FUNCTION_BLOCK FbGSS (* Генератор сигналов и псевдослучайных чисел. *)
  (* Standard: 61499-1; Description: Генератор сигналов и псевдослучайных чисел. Simple FB with one algorithm *)
  (* Version 2.1, 2026-03-20, VA, LIB_PLC *)
  (* Documentation:
  // Генератор сигналов и псевдослучайных чисел. //             DbGSS //     +--------------------+ //     |       FbGSS        | //    -|Amplitude       Sine|->- //    -|Period        Cosine|->- //    -|Phase     RectangleR|->- //    -|Offset    RectangleB|->- //    -|PulseTime   Triangle|->- //    -|Ts              Prnd|->- //     +--------------------+
  *)
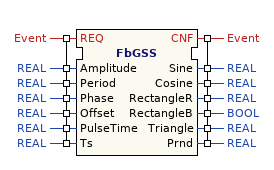
  EVENT_INPUT
    REQ WITH Amplitude, Period, Phase, Offset, PulseTime, Ts; (* Normal Execution Request *)
  END_EVENT
  EVENT_OUTPUT
    CNF WITH Sine, Cosine, RectangleR, RectangleB, Triangle, Prnd; (* Execution Confirmation *)
  END_EVENT
  VAR_INPUT
    Amplitude : REAL := 1.0; (* Амплитуда выходного сигнала. *)
    Period : REAL := 10.0; (* Период выходного сигнала [с]. *)
    Phase : REAL := 0.0; (* Фаза выходного сигнала [рад]. *)
    Offset : REAL := 0.0; (* Постоянная составляющая выходного сигнала. *)
    PulseTime : REAL := 5.0; (* Время импульса [с]. *)
    Ts : REAL := 0.1; (* Шаг дискретизации по времени [с]. *)
  END_VAR
  VAR_OUTPUT
    Sine : REAL := 0.0; (* Синусоидальный сигнал. *)
    Cosine : REAL := 0.0; (* Косинусоидальный сигнал. *)
    RectangleR : REAL := 0.0; (* Прямоугольный сигнал вещественный. *)
    RectangleB : BOOL := FALSE; (* Прямоугольный сигнал булевый. *)
    Triangle : REAL := 0.0; (* Треугольный, линейно нарастающий и убывающий сигнал. *)
    Prnd : REAL := 0.0; (* Псевдослучайные числа в диапазоне 0...1. *)
  END_VAR
  VAR CONSTANT
    PI : REAL := 3.14159265358979323846; (* Число Пи. *)
  END_VAR
  VAR
    CurrentTime : REAL := 0.0;
    IntegratorTriangle : REAL := 0.0;
    SummatorRnd : DINT := 1;
    Tmp : DWORD := 16#00000000;
  END_VAR
  EC_STATES
    REQ : REQ -> CNF;
  END_STATES
  ALGORITHM REQ IN ST:
Sine := Amplitude * SIN(2.0 * PI * (1.0 / Period) * CurrentTime + Phase) + Offset;
Cosine := Amplitude * COS(2.0 * PI * (1.0 / Period) * CurrentTime + Phase) + Offset;

IF (CurrentTime < PulseTime) THEN // Прямоугольные импульсы.
	RectangleR := Amplitude + Offset;
	RectangleB := TRUE;
ELSE
	RectangleR := Offset;
	RectangleB := FALSE;
END_IF;

IF (CurrentTime <= (Period * 0.5)) THEN // Треугольные импульсы.
	IntegratorTriangle := IntegratorTriangle + Ts;
ELSE
	IntegratorTriangle := IntegratorTriangle - Ts;
END_IF;
IF (Period <> 0.0) THEN
	Triangle := (((IntegratorTriangle * 2.0) / Period) * Amplitude) + Offset;
END_IF;

// Псевдослучайные числа линейный конгруэнтный метод.
SummatorRnd := SummatorRnd * 1103515245 + 12345;
// Принудительно отбрасывающей младшие 16 и один старший разряд.
Tmp := DINT_TO_DWORD(SummatorRnd) AND 2#01111111111111110000000000000000;
// Арифметический сдвиг вправо на 16бит.
Tmp := SHR(Tmp, 16);
// Масштабирование 0...32767 -> 0...1
Prnd := (DINT_TO_REAL(DWORD_TO_DINT(Tmp)) / 32767.0) * Amplitude + Offset;

CurrentTime := CurrentTime + Ts; // Формирование периода.
IF (CurrentTime >= Period) THEN
	CurrentTime := 0.0;
	IntegratorTriangle := 0.0;
END_IF;

// @COPYLEFT ALL WRONGS RESERVED :)
// Author: VA
// Contacts: DIY.PLC.314@gmail.com
// Date start LIB_PLC: 2014
// License: GNU GPL-2.0-or-later
// https://www.gnu.org/licenses/old-licenses/gpl-2.0.html
// https://www.youtube.com/watch?v=n1F_MfLRlX0
// https://www.youtube.com/@DIY_PLC
// https://github.com/DIYPLC/LIB_PLC
// https://oshwlab.com/diy.plc.314/PLC_HW1_SW1
// https://3dtoday.ru/3d-models/mechanical-parts/body/korpus-na-din-reiku
// https://t.me/DIY_PLC
  END_ALGORITHM
END_FUNCTION_BLOCK
